Fanuc KAREL source: kt00518.KL

-- PROVISIONAL review KL for V1013-1; original PC SHA256 17d66d2836c536c76518f5fa5d95ef52d623d8f4397dedd6bfc4e027cd64b8d4
-- Incomplete behavior may be omitted. Consult companion uncertainty JSON. Do not deploy.
PROGRAM KT00518
%NOLOCKGROUP
VAR
  OUT : BOOLEAN
-- UNRESOLVED_DECL P1 type=000106
-- UNRESOLVED_DECL P2 type=000102
BEGIN
  -- UNRESOLVED_PC offsets 5-20; opcodes 2E,22,32,35
  -- UNRESOLVED_PC offsets 25-40; opcodes 2E,22,32,35
  -- UNRESOLVED_PC offsets 45-78; opcodes 49,7E,49,7E,AC,23
  -- UNRESOLVED_PC offsets 83-87; opcodes 7F
END KT00518
